// TwinCAT 3 PLC project SaftyPLC
// ProgramVersion: 3.1.4026.13
// libraries:
//   Tc2_Standard, * (Beckhoff Automation GmbH)
//   Tc2_System, * (Beckhoff Automation GmbH)
//   Tc2_Utilities, * (Beckhoff Automation GmbH)
//   Tc3_EventLogger, * (Beckhoff Automation GmbH)
//   Tc3_Module, * (Beckhoff Automation GmbH)
// project tree:
//   GVLs/ GVL_IO.TcGVL (not stored), GVL_Safety.TcGVL
//   / PlcTask.TcTTO
//   POUs/ MAIN.TcPOU
// real-time tasks:
//   TASK XTS Task: cycle T#500us, priority 1, ADS port 350
//   TASK Job Task: cycle default, priority 32
//   TASK MC-Task (MET): cycle T#2ms, priority 3, ADS port 521
//   TASK MC-Task (MPT): cycle T#10ms, priority 8, ADS port 531
//   TASK PlcTask: cycle T#500us, priority 20, ADS port 351
// motion (NC):
//   TASK NC-Task 1 SAF: cycle T#2ms, priority 4, ADS port 501
//   TASK NC-Task 1 SVB: cycle T#10ms, priority 9, ADS port 511
//   AXIS Axis 1 (id 1)
//     Velo: Maximum=4000
//     OtherSettings: AllowMotionCmdToSlave=true
//     encoder EncType=28
//       EncPara: MaxCount=#xffffffff
//     drive DrvType=22
//       DrvPara: MaxCount=#xffffffff, DriveControlDWord=#x00000100
//         Analog: VeloReferenz=4200, TorqueSetpointScale=10, ScaleFactorActTorque=0.1
//         TimeComp: TaskDelayCycles=1
//     controller CtrType=1
//       CtrPara: PriorControlFactor=1
//         Observer: BandWidth=20
// I/O:
//   DEVICE Device 8 (EtherCAT), AmsNetId 0.0.0.0.9.1
//     Box 77 (AT5100-0100) [AT5100-0100 XTS XL, TwinSAFE]
//       modules: Module 1 (SAFETY)
//     Box 78 (AT5100-0100) [AT5100-0100 XTS XL, TwinSAFE]
//       modules: Module 1 (SAFETY)
//     Box 79 (AT5100-0100) [AT5100-0100 XTS XL, TwinSAFE]
//       modules: Module 1 (SAFETY)
//     Box 80 (AT5100-0100) [AT5100-0100 XTS XL, TwinSAFE]
//       modules: Module 1 (SAFETY)
//     Box 81 (AT5100-0100) [AT5100-0100 XTS XL, TwinSAFE]
//       modules: Module 1 (SAFETY)
//     Box 18 (AT5100-0100) [AT5100-0100 XTS XL, TwinSAFE]
//       modules: Module 1 (SAFETY)
//     Box 19 (AT5100-0100) [AT5100-0100 XTS XL, TwinSAFE]
//       modules: Module 1 (SAFETY)
//     Box 20 (AT5100-0100) [AT5100-0100 XTS XL, TwinSAFE]
//       modules: Module 1 (SAFETY)
//     Box 21 (AT5100-0100) [AT5100-0100 XTS XL, TwinSAFE]
//       modules: Module 1 (SAFETY)
//     Box 22 (AT5100-0100) [AT5100-0100 XTS XL, TwinSAFE]
//       modules: Module 1 (SAFETY)
//   DEVICE Device 1 (EtherCAT), AmsNetId 0.0.0.0.2.1
//     Term 1 (EK1200) [EK1200-5000 EtherCAT Power supply (2A E-Bus)]
//       Term 2 (EL1809) [EL1809 16Ch. Dig. Input 24V, 3ms]
//       Term 3 (EL2809) [EL2809 16Ch. Dig. Output 24V, 0.5A]
//       Term 4 (EL1918) [EL1918, 8Ch. Safety Input 24V, TwinSAFE]
//         modules: Module 2 (FSLOGIC)
//       Term 5 (EK1110) [EK1110 EtherCAT extension]
//     Box 11 (Drive1211) [Drive1211]
//       modules: Module 1 (Standard Process Data)
//   DEVICE Device 2 (EtherCAT Automation Protocol), AmsNetId 0.0.0.0.3.1
//     Box 28 (Publisher)
//     Box 29 (Subscriber)
// variable links:
//   Device 1 (EtherCAT) <-> Device 2 (EtherCAT Automation Protocol)/Box 28 (Publisher)
//     Term 1 (EK1200)/Term 4 (EL1918)/ConnectionInputs/Message_144 TxPDO <-> Safety/Outputs/VarData
//   Device 1 (EtherCAT) <-> Device 2 (EtherCAT Automation Protocol)/Box 29 (Subscriber)
//     Term 1 (EK1200)/Term 4 (EL1918)/ConnectionOutputs/Message_144 RxPDO <-> Safety/Inputs/VarData
//   Device 2 (EtherCAT Automation Protocol) <-> MC Project IPC2/Groups/IPC 2 In Connection
//     Box 28 (Publisher)/MC Track - XL In Syst 2/Outputs/VarData <-> McToMc/ToNeighbourSystem
//     Box 29 (Subscriber)/MC Track - XL Out Syst 1/Inputs/VarData <-> McToMc/FromNeighbourSystem
//   Device 2 (EtherCAT Automation Protocol) <-> MC Project IPC2/Groups/IPC 2 Out Connection
//     Box 28 (Publisher)/MC Track - XL Out Syst 2/Outputs/VarData <-> McToMc/ToNeighbourSystem
//     Box 29 (Subscriber)/MC Track - XL In Syst 1/Inputs/VarData <-> McToMc/FromNeighbourSystem
//   Device 8 (EtherCAT) <-> Device 1 (EtherCAT)/Term 1 (EK1200)/Term 4 (EL1918)
//     Box 18 (AT5100-0100)/Module 1 (SAFETY)/SAFETY FSoE Connection 1 Receive Message/Message_4 <-> ConnectionInputs/Message_71 TxPDO
//     Box 19 (AT5100-0100)/Module 1 (SAFETY)/SAFETY FSoE Connection 1 Receive Message/Message_4 <-> ConnectionInputs/Message_76 TxPDO
//     Box 20 (AT5100-0100)/Module 1 (SAFETY)/SAFETY FSoE Connection 1 Receive Message/Message_4 <-> ConnectionInputs/Message_77 TxPDO
//     Box 21 (AT5100-0100)/Module 1 (SAFETY)/SAFETY FSoE Connection 1 Receive Message/Message_4 <-> ConnectionInputs/Message_78 TxPDO
//     Box 22 (AT5100-0100)/Module 1 (SAFETY)/SAFETY FSoE Connection 1 Receive Message/Message_4 <-> ConnectionInputs/Message_79 TxPDO
//     Box 77 (AT5100-0100)/Module 1 (SAFETY)/SAFETY FSoE Connection 1 Receive Message/Message_4 <-> ConnectionInputs/Message_134 TxPDO
//     Box 78 (AT5100-0100)/Module 1 (SAFETY)/SAFETY FSoE Connection 1 Receive Message/Message_4 <-> ConnectionInputs/Message_135 TxPDO
//     Box 79 (AT5100-0100)/Module 1 (SAFETY)/SAFETY FSoE Connection 1 Receive Message/Message_4 <-> ConnectionInputs/Message_136 TxPDO
//     Box 80 (AT5100-0100)/Module 1 (SAFETY)/SAFETY FSoE Connection 1 Receive Message/Message_4 <-> ConnectionInputs/Message_137 TxPDO
//     Box 81 (AT5100-0100)/Module 1 (SAFETY)/SAFETY FSoE Connection 1 Receive Message/Message_4 <-> ConnectionInputs/Message_138 TxPDO
//     Box 18 (AT5100-0100)/Module 1 (SAFETY)/SAFETY FSoE Connection 1 Send Message/Message_4 <-> ConnectionOutputs/Message_71 RxPDO
//     Box 19 (AT5100-0100)/Module 1 (SAFETY)/SAFETY FSoE Connection 1 Send Message/Message_4 <-> ConnectionOutputs/Message_76 RxPDO
//     Box 20 (AT5100-0100)/Module 1 (SAFETY)/SAFETY FSoE Connection 1 Send Message/Message_4 <-> ConnectionOutputs/Message_77 RxPDO
//     Box 21 (AT5100-0100)/Module 1 (SAFETY)/SAFETY FSoE Connection 1 Send Message/Message_4 <-> ConnectionOutputs/Message_78 RxPDO
//     Box 22 (AT5100-0100)/Module 1 (SAFETY)/SAFETY FSoE Connection 1 Send Message/Message_4 <-> ConnectionOutputs/Message_79 RxPDO
//     Box 77 (AT5100-0100)/Module 1 (SAFETY)/SAFETY FSoE Connection 1 Send Message/Message_4 <-> ConnectionOutputs/Message_134 RxPDO
//     Box 78 (AT5100-0100)/Module 1 (SAFETY)/SAFETY FSoE Connection 1 Send Message/Message_4 <-> ConnectionOutputs/Message_135 RxPDO
//     Box 79 (AT5100-0100)/Module 1 (SAFETY)/SAFETY FSoE Connection 1 Send Message/Message_4 <-> ConnectionOutputs/Message_136 RxPDO
//     Box 80 (AT5100-0100)/Module 1 (SAFETY)/SAFETY FSoE Connection 1 Send Message/Message_4 <-> ConnectionOutputs/Message_137 RxPDO
//     Box 81 (AT5100-0100)/Module 1 (SAFETY)/SAFETY FSoE Connection 1 Send Message/Message_4 <-> ConnectionOutputs/Message_138 RxPDO
//   MC Project IPC2/Axes/MC_Mover 01 IPC2 <-> MC Project IPC2/Axes/MC_Mover 01 IPC2/XConverter 01 IPC2
//     IoToMc/STD <-> OutputsToMC3/HWToMC3
//     McToIo/STD <-> InputsFromPlanarMover/MC3ToHW
//   MC Project IPC2/Axes/MC_Mover 02 IPC2 <-> MC Project IPC2/Axes/MC_Mover 02 IPC2/XConverter 02 IPC2
//     IoToMc/STD <-> OutputsToMC3/HWToMC3
//     McToIo/STD <-> InputsFromPlanarMover/MC3ToHW
//   MC Project IPC2/Axes/MC_Mover 03 IPC2 <-> MC Project IPC2/Axes/MC_Mover 03 IPC2/XConverter 03 IPC2
//     IoToMc/STD <-> OutputsToMC3/HWToMC3
//     McToIo/STD <-> InputsFromPlanarMover/MC3ToHW
//   MC Project IPC2/Axes/MC_Mover 04 IPC2 <-> MC Project IPC2/Axes/MC_Mover 04 IPC2/XConverter 04 IPC2
//     IoToMc/STD <-> OutputsToMC3/HWToMC3
//     McToIo/STD <-> InputsFromPlanarMover/MC3ToHW
//   MC Project IPC2/Axes/MC_Mover 05 IPC2 <-> MC Project IPC2/Axes/MC_Mover 05 IPC2/XConverter 05 IPC2
//     IoToMc/STD <-> OutputsToMC3/HWToMC3
//     McToIo/STD <-> InputsFromPlanarMover/MC3ToHW
//   MC Project IPC2/Axes/MC_Mover 06 IPC2 <-> MC Project IPC2/Axes/MC_Mover 06 IPC2/XConverter 06 IPC2
//     IoToMc/STD <-> OutputsToMC3/HWToMC3
//     McToIo/STD <-> InputsFromPlanarMover/MC3ToHW
//   MC Project IPC2/Axes/MC_Mover 07 IPC2 <-> MC Project IPC2/Axes/MC_Mover 07 IPC2/XConverter 07 IPC2
//     IoToMc/STD <-> OutputsToMC3/HWToMC3
//     McToIo/STD <-> InputsFromPlanarMover/MC3ToHW
//   MC Project IPC2/Axes/MC_Mover 08 IPC2 <-> MC Project IPC2/Axes/MC_Mover 08 IPC2/XConverter 08 IPC2
//     IoToMc/STD <-> OutputsToMC3/HWToMC3
//     McToIo/STD <-> InputsFromPlanarMover/MC3ToHW
//   MC Project IPC2/Axes/MC_Mover 09 IPC2 <-> MC Project IPC2/Axes/MC_Mover 09 IPC2/XConverter 09 IPC2
//     IoToMc/STD <-> OutputsToMC3/HWToMC3
//     McToIo/STD <-> InputsFromPlanarMover/MC3ToHW
//   MC Project IPC2/Axes/MC_Mover 10 IPC2 <-> MC Project IPC2/Axes/MC_Mover 10 IPC2/XConverter 10 IPC2
//     IoToMc/STD <-> OutputsToMC3/HWToMC3
//     McToIo/STD <-> InputsFromPlanarMover/MC3ToHW
//   MC Project IPC2/Axes/MC_Mover 11 IPC2 <-> MC Project IPC2/Axes/MC_Mover 11 IPC2/XConverter 11 IPC2
//     IoToMc/STD <-> OutputsToMC3/HWToMC3
//     McToIo/STD <-> InputsFromPlanarMover/MC3ToHW
//   MC Project IPC2/Axes/MC_Mover 12 IPC2 <-> MC Project IPC2/Axes/MC_Mover 12 IPC2/XConverter 12 IPC2
//     IoToMc/STD <-> OutputsToMC3/HWToMC3
//     McToIo/STD <-> InputsFromPlanarMover/MC3ToHW
//   MC3_Multi_IPC2/MC3_Multi_IPC2 Instance <-> Device 2 (EtherCAT Automation Protocol)/Box 29 (Subscriber)
//     PlcTask Inputs/GVL_DataExchange.Dynamics <-> Command/Inputs/VarData/Dynamics
//   MC3_Multi_IPC2/MC3_Multi_IPC2 Instance <-> MC Project IPC2/Axes/MC_Mover 01 IPC2
//     PlcTask Inputs/GVL_MC.fbMover[1].fbPlanarMover.MCTOPLC/ACT <-> McToPlc/ACT
//     PlcTask Inputs/GVL_MC.fbMover[1].fbPlanarMover.MCTOPLC/COORDMODE <-> McToPlc/COORDMODE
//     PlcTask Inputs/GVL_MC.fbMover[1].fbPlanarMover.MCTOPLC/SET <-> McToPlc/SET
//     PlcTask Inputs/GVL_MC.fbMover[1].fbPlanarMover.MCTOPLC/SETONTRACK <-> McToPlc/SETONTRACK
//     PlcTask Inputs/GVL_MC.fbMover[1].fbPlanarMover.MCTOPLC/STD <-> McToPlc/STD
//     PlcTask Outputs/GVL_MC.fbMover[1].fbPlanarMover.PLCTOMC/STD <-> PlcToMc/STD
//   MC3_Multi_IPC2/MC3_Multi_IPC2 Instance <-> MC Project IPC2/Axes/MC_Mover 02 IPC2
//     PlcTask Inputs/GVL_MC.fbMover[2].fbPlanarMover.MCTOPLC/ACT <-> McToPlc/ACT
//     PlcTask Inputs/GVL_MC.fbMover[2].fbPlanarMover.MCTOPLC/COORDMODE <-> McToPlc/COORDMODE
//     PlcTask Inputs/GVL_MC.fbMover[2].fbPlanarMover.MCTOPLC/SET <-> McToPlc/SET
//     PlcTask Inputs/GVL_MC.fbMover[2].fbPlanarMover.MCTOPLC/SETONTRACK <-> McToPlc/SETONTRACK
//     PlcTask Inputs/GVL_MC.fbMover[2].fbPlanarMover.MCTOPLC/STD <-> McToPlc/STD
//     PlcTask Outputs/GVL_MC.fbMover[2].fbPlanarMover.PLCTOMC/STD <-> PlcToMc/STD
//   MC3_Multi_IPC2/MC3_Multi_IPC2 Instance <-> MC Project IPC2/Axes/MC_Mover 03 IPC2
//     PlcTask Inputs/GVL_MC.fbMover[3].fbPlanarMover.MCTOPLC/ACT <-> McToPlc/ACT
//     PlcTask Inputs/GVL_MC.fbMover[3].fbPlanarMover.MCTOPLC/COORDMODE <-> McToPlc/COORDMODE
//     PlcTask Inputs/GVL_MC.fbMover[3].fbPlanarMover.MCTOPLC/SET <-> McToPlc/SET
//     PlcTask Inputs/GVL_MC.fbMover[3].fbPlanarMover.MCTOPLC/SETONTRACK <-> McToPlc/SETONTRACK
//     PlcTask Inputs/GVL_MC.fbMover[3].fbPlanarMover.MCTOPLC/STD <-> McToPlc/STD
//     PlcTask Outputs/GVL_MC.fbMover[3].fbPlanarMover.PLCTOMC/STD <-> PlcToMc/STD
//   MC3_Multi_IPC2/MC3_Multi_IPC2 Instance <-> MC Project IPC2/Axes/MC_Mover 04 IPC2
//     PlcTask Inputs/GVL_MC.fbMover[4].fbPlanarMover.MCTOPLC/ACT <-> McToPlc/ACT
//     PlcTask Inputs/GVL_MC.fbMover[4].fbPlanarMover.MCTOPLC/COORDMODE <-> McToPlc/COORDMODE
//     PlcTask Inputs/GVL_MC.fbMover[4].fbPlanarMover.MCTOPLC/SET <-> McToPlc/SET
//     PlcTask Inputs/GVL_MC.fbMover[4].fbPlanarMover.MCTOPLC/SETONTRACK <-> McToPlc/SETONTRACK
//     PlcTask Inputs/GVL_MC.fbMover[4].fbPlanarMover.MCTOPLC/STD <-> McToPlc/STD
//     PlcTask Outputs/GVL_MC.fbMover[4].fbPlanarMover.PLCTOMC/STD <-> PlcToMc/STD
//   MC3_Multi_IPC2/MC3_Multi_IPC2 Instance <-> MC Project IPC2/Axes/MC_Mover 05 IPC2
//     PlcTask Inputs/GVL_MC.fbMover[5].fbPlanarMover.MCTOPLC/ACT <-> McToPlc/ACT
//     PlcTask Inputs/GVL_MC.fbMover[5].fbPlanarMover.MCTOPLC/COORDMODE <-> McToPlc/COORDMODE
//     PlcTask Inputs/GVL_MC.fbMover[5].fbPlanarMover.MCTOPLC/SET <-> McToPlc/SET
//     PlcTask Inputs/GVL_MC.fbMover[5].fbPlanarMover.MCTOPLC/SETONTRACK <-> McToPlc/SETONTRACK
//     PlcTask Inputs/GVL_MC.fbMover[5].fbPlanarMover.MCTOPLC/STD <-> McToPlc/STD
//     PlcTask Outputs/GVL_MC.fbMover[5].fbPlanarMover.PLCTOMC/STD <-> PlcToMc/STD
//   MC3_Multi_IPC2/MC3_Multi_IPC2 Instance <-> MC Project IPC2/Axes/MC_Mover 06 IPC2
//     PlcTask Inputs/GVL_MC.fbMover[6].fbPlanarMover.MCTOPLC/ACT <-> McToPlc/ACT
//     PlcTask Inputs/GVL_MC.fbMover[6].fbPlanarMover.MCTOPLC/COORDMODE <-> McToPlc/COORDMODE
//     PlcTask Inputs/GVL_MC.fbMover[6].fbPlanarMover.MCTOPLC/SET <-> McToPlc/SET
//     PlcTask Inputs/GVL_MC.fbMover[6].fbPlanarMover.MCTOPLC/SETONTRACK <-> McToPlc/SETONTRACK
//     PlcTask Inputs/GVL_MC.fbMover[6].fbPlanarMover.MCTOPLC/STD <-> McToPlc/STD
//     PlcTask Outputs/GVL_MC.fbMover[6].fbPlanarMover.PLCTOMC/STD <-> PlcToMc/STD
//   MC3_Multi_IPC2/MC3_Multi_IPC2 Instance <-> MC Project IPC2/Axes/MC_Mover 07 IPC2
//     PlcTask Inputs/GVL_MC.fbMover[7].fbPlanarMover.MCTOPLC/ACT <-> McToPlc/ACT
//     PlcTask Inputs/GVL_MC.fbMover[7].fbPlanarMover.MCTOPLC/COORDMODE <-> McToPlc/COORDMODE
//     PlcTask Inputs/GVL_MC.fbMover[7].fbPlanarMover.MCTOPLC/SET <-> McToPlc/SET
//     PlcTask Inputs/GVL_MC.fbMover[7].fbPlanarMover.MCTOPLC/SETONTRACK <-> McToPlc/SETONTRACK
//     PlcTask Inputs/GVL_MC.fbMover[7].fbPlanarMover.MCTOPLC/STD <-> McToPlc/STD
//     PlcTask Outputs/GVL_MC.fbMover[7].fbPlanarMover.PLCTOMC/STD <-> PlcToMc/STD
//   MC3_Multi_IPC2/MC3_Multi_IPC2 Instance <-> MC Project IPC2/Axes/MC_Mover 08 IPC2
//     PlcTask Inputs/GVL_MC.fbMover[8].fbPlanarMover.MCTOPLC/ACT <-> McToPlc/ACT
//     PlcTask Inputs/GVL_MC.fbMover[8].fbPlanarMover.MCTOPLC/COORDMODE <-> McToPlc/COORDMODE
//     PlcTask Inputs/GVL_MC.fbMover[8].fbPlanarMover.MCTOPLC/SET <-> McToPlc/SET
//     PlcTask Inputs/GVL_MC.fbMover[8].fbPlanarMover.MCTOPLC/SETONTRACK <-> McToPlc/SETONTRACK
//     PlcTask Inputs/GVL_MC.fbMover[8].fbPlanarMover.MCTOPLC/STD <-> McToPlc/STD
//     PlcTask Outputs/GVL_MC.fbMover[8].fbPlanarMover.PLCTOMC/STD <-> PlcToMc/STD
//   MC3_Multi_IPC2/MC3_Multi_IPC2 Instance <-> MC Project IPC2/Axes/MC_Mover 09 IPC2
//     PlcTask Inputs/GVL_MC.fbMover[9].fbPlanarMover.MCTOPLC/ACT <-> McToPlc/ACT
//     PlcTask Inputs/GVL_MC.fbMover[9].fbPlanarMover.MCTOPLC/COORDMODE <-> McToPlc/COORDMODE
//     PlcTask Inputs/GVL_MC.fbMover[9].fbPlanarMover.MCTOPLC/SET <-> McToPlc/SET
//     PlcTask Inputs/GVL_MC.fbMover[9].fbPlanarMover.MCTOPLC/SETONTRACK <-> McToPlc/SETONTRACK
//     PlcTask Inputs/GVL_MC.fbMover[9].fbPlanarMover.MCTOPLC/STD <-> McToPlc/STD
//     PlcTask Outputs/GVL_MC.fbMover[9].fbPlanarMover.PLCTOMC/STD <-> PlcToMc/STD
//   MC3_Multi_IPC2/MC3_Multi_IPC2 Instance <-> MC Project IPC2/Axes/MC_Mover 10 IPC2
//     PlcTask Inputs/GVL_MC.fbMover[10].fbPlanarMover.MCTOPLC/ACT <-> McToPlc/ACT
//     PlcTask Inputs/GVL_MC.fbMover[10].fbPlanarMover.MCTOPLC/COORDMODE <-> McToPlc/COORDMODE
//     PlcTask Inputs/GVL_MC.fbMover[10].fbPlanarMover.MCTOPLC/SET <-> McToPlc/SET
//     PlcTask Inputs/GVL_MC.fbMover[10].fbPlanarMover.MCTOPLC/SETONTRACK <-> McToPlc/SETONTRACK
//     PlcTask Inputs/GVL_MC.fbMover[10].fbPlanarMover.MCTOPLC/STD <-> McToPlc/STD
//     PlcTask Outputs/GVL_MC.fbMover[10].fbPlanarMover.PLCTOMC/STD <-> PlcToMc/STD
//   MC3_Multi_IPC2/MC3_Multi_IPC2 Instance <-> MC Project IPC2/Axes/MC_Mover 11 IPC2
//     PlcTask Inputs/GVL_MC.fbMover[11].fbPlanarMover.MCTOPLC/ACT <-> McToPlc/ACT
//     PlcTask Inputs/GVL_MC.fbMover[11].fbPlanarMover.MCTOPLC/COORDMODE <-> McToPlc/COORDMODE
//     PlcTask Inputs/GVL_MC.fbMover[11].fbPlanarMover.MCTOPLC/SET <-> McToPlc/SET
//     PlcTask Inputs/GVL_MC.fbMover[11].fbPlanarMover.MCTOPLC/SETONTRACK <-> McToPlc/SETONTRACK
//     PlcTask Inputs/GVL_MC.fbMover[11].fbPlanarMover.MCTOPLC/STD <-> McToPlc/STD
//     PlcTask Outputs/GVL_MC.fbMover[11].fbPlanarMover.PLCTOMC/STD <-> PlcToMc/STD
//   MC3_Multi_IPC2/MC3_Multi_IPC2 Instance <-> MC Project IPC2/Axes/MC_Mover 12 IPC2
//     PlcTask Inputs/GVL_MC.fbMover[12].fbPlanarMover.MCTOPLC/ACT <-> McToPlc/ACT
//     PlcTask Inputs/GVL_MC.fbMover[12].fbPlanarMover.MCTOPLC/COORDMODE <-> McToPlc/COORDMODE
//     PlcTask Inputs/GVL_MC.fbMover[12].fbPlanarMover.MCTOPLC/SET <-> McToPlc/SET
//     PlcTask Inputs/GVL_MC.fbMover[12].fbPlanarMover.MCTOPLC/SETONTRACK <-> McToPlc/SETONTRACK
//     PlcTask Inputs/GVL_MC.fbMover[12].fbPlanarMover.MCTOPLC/STD <-> McToPlc/STD
//     PlcTask Outputs/GVL_MC.fbMover[12].fbPlanarMover.PLCTOMC/STD <-> PlcToMc/STD
//   MC3_Multi_IPC2/MC3_Multi_IPC2 Instance <-> MC Project IPC2/Groups/IPC 2 In Connection
//     PlcTask Inputs/GVL_MC.EnterSystem.MCTOPLC_STD <-> McToPlc/STD
//   MC3_Multi_IPC2/MC3_Multi_IPC2 Instance <-> MC Project IPC2/Groups/IPC 2 Out Connection
//     PlcTask Inputs/GVL_MC.ExitSystem.MCTOPLC_STD <-> McToPlc/STD
//   MC3_Multi_IPC2/MC3_Multi_IPC2 Instance <-> MC Project IPC2/Groups/McTrack1
//     PlcTask Inputs/GVL_MC.aMcTracks[1].MCTOPLC_STD <-> McToPlc/STD
//   SaftyPLC/SaftyPLC Instance <-> Device 1 (EtherCAT)/Box 11 (Drive1211)
//     PlcTask Inputs/GVL_IO.StatusDrive1121 <-> Module 1 (Standard Process Data)/TxPDO1Map entries/Statusword
//     PlcTask Inputs/GVL_IO.VoltageAct <-> Module 1 (Standard Process Data)/TxPDO1Map entries/Zwischenkreisspannung
//     PlcTask Outputs/GVL_IO.ControlDrive1121 <-> Module 1 (Standard Process Data)/RxPDO1Map entries/Controlword
//     PlcTask Outputs/GVL_IO.VoltageSet <-> Module 1 (Standard Process Data)/RxPDO1Map entries/Zwischenkreisspannung Soll
//   SaftyPLC/SaftyPLC Instance <-> Device 1 (EtherCAT)/Term 1 (EK1200)/Term 2 (EL1809)
//     PlcTask Inputs/GVL_Safety.HWReset <-> Channel 16/Input
//     PlcTask Inputs/GVL_Safety.HWStart <-> Channel 14/Input
//     PlcTask Inputs/GVL_Safety.HWStop <-> Channel 15/Input
//   SaftyPLC/SaftyPLC Instance <-> Device 1 (EtherCAT)/Term 1 (EK1200)/Term 3 (EL2809)
//     PlcTask Outputs/GVL_Safety.HWSafetyOk <-> Channel 14/Output
//     PlcTask Outputs/GVL_Safety.HWerror <-> Channel 15/Output
//   SaftyPLC/SaftyPLC Instance <-> Device 1 (EtherCAT)/Term 1 (EK1200)/Term 4 (EL1918)
//     PlcTask Inputs/GVL_Safety.SaeftyOk <-> StandardInputs/Standard Out Var 139
//     PlcTask Outputs/GVL_Safety.Reset <-> StandardOutputs/Standard In Var 1
//     PlcTask Outputs/GVL_Safety.Run <-> StandardOutputs/Standard In Var 2
//     PlcTask Outputs/GVL_Safety.Start <-> StandardOutputs/Standard In Var 140
//     PlcTask Outputs/GVL_Safety.Start <-> StandardOutputs/Standard In Var 75
//   SaftyPLC/SaftyPLC Instance <-> Device 2 (EtherCAT Automation Protocol)/Box 29 (Subscriber)
//     PlcTask Inputs/GVL_Safety.MasterReset <-> Command/Inputs/VarData/Reset
//     PlcTask Inputs/GVL_Safety.SafetyInRun <-> Command/Inputs/VarData/Run
//   SaftyPLC/SaftyPLC Instance <-> Device 8 (EtherCAT)/Box 18 (AT5100-0100)
//     PlcTask Outputs/GVL_Safety.Reset <-> Module 1 (SAFETY)/SAFETY Standard Outputdata/Standard In Var 1
//     PlcTask Outputs/GVL_Safety.Run <-> Module 1 (SAFETY)/SAFETY Standard Outputdata/Standard In Var 2
//   SaftyPLC/SaftyPLC Instance <-> Device 8 (EtherCAT)/Box 19 (AT5100-0100)
//     PlcTask Outputs/GVL_Safety.Reset <-> Module 1 (SAFETY)/SAFETY Standard Outputdata/Standard In Var 1
//     PlcTask Outputs/GVL_Safety.Run <-> Module 1 (SAFETY)/SAFETY Standard Outputdata/Standard In Var 2
//   SaftyPLC/SaftyPLC Instance <-> Device 8 (EtherCAT)/Box 20 (AT5100-0100)
//     PlcTask Outputs/GVL_Safety.Reset <-> Module 1 (SAFETY)/SAFETY Standard Outputdata/Standard In Var 1
//     PlcTask Outputs/GVL_Safety.Run <-> Module 1 (SAFETY)/SAFETY Standard Outputdata/Standard In Var 2
//   SaftyPLC/SaftyPLC Instance <-> Device 8 (EtherCAT)/Box 21 (AT5100-0100)
//     PlcTask Outputs/GVL_Safety.Reset <-> Module 1 (SAFETY)/SAFETY Standard Outputdata/Standard In Var 1
//     PlcTask Outputs/GVL_Safety.Run <-> Module 1 (SAFETY)/SAFETY Standard Outputdata/Standard In Var 2
//   SaftyPLC/SaftyPLC Instance <-> Device 8 (EtherCAT)/Box 22 (AT5100-0100)
//     PlcTask Outputs/GVL_Safety.Reset <-> Module 1 (SAFETY)/SAFETY Standard Outputdata/Standard In Var 1
//     PlcTask Outputs/GVL_Safety.Run <-> Module 1 (SAFETY)/SAFETY Standard Outputdata/Standard In Var 2
//   SaftyPLC/SaftyPLC Instance <-> Device 8 (EtherCAT)/Box 77 (AT5100-0100)
//     PlcTask Outputs/GVL_Safety.Reset <-> Module 1 (SAFETY)/SAFETY Standard Outputdata/Standard In Var 1
//     PlcTask Outputs/GVL_Safety.Run <-> Module 1 (SAFETY)/SAFETY Standard Outputdata/Standard In Var 2
//   SaftyPLC/SaftyPLC Instance <-> Device 8 (EtherCAT)/Box 78 (AT5100-0100)
//     PlcTask Outputs/GVL_Safety.Reset <-> Module 1 (SAFETY)/SAFETY Standard Outputdata/Standard In Var 1
//     PlcTask Outputs/GVL_Safety.Run <-> Module 1 (SAFETY)/SAFETY Standard Outputdata/Standard In Var 2
//   SaftyPLC/SaftyPLC Instance <-> Device 8 (EtherCAT)/Box 79 (AT5100-0100)
//     PlcTask Outputs/GVL_Safety.Reset <-> Module 1 (SAFETY)/SAFETY Standard Outputdata/Standard In Var 1
//     PlcTask Outputs/GVL_Safety.Run <-> Module 1 (SAFETY)/SAFETY Standard Outputdata/Standard In Var 2
//   SaftyPLC/SaftyPLC Instance <-> Device 8 (EtherCAT)/Box 80 (AT5100-0100)
//     PlcTask Outputs/GVL_Safety.Reset <-> Module 1 (SAFETY)/SAFETY Standard Outputdata/Standard In Var 1
//     PlcTask Outputs/GVL_Safety.Run <-> Module 1 (SAFETY)/SAFETY Standard Outputdata/Standard In Var 2
//   SaftyPLC/SaftyPLC Instance <-> Device 8 (EtherCAT)/Box 81 (AT5100-0100)
//     PlcTask Outputs/GVL_Safety.Reset <-> Module 1 (SAFETY)/SAFETY Standard Outputdata/Standard In Var 1
//     PlcTask Outputs/GVL_Safety.Run <-> Module 1 (SAFETY)/SAFETY Standard Outputdata/Standard In Var 2
//   (this object) <-> TcCOM Objects/XTS ProcessingUnit 2/XL Part Main/XL Module 10
//     Box 19 (AT5100-0100)/DRV Commutation angle/Commutation angle <-> Data Pointer/CommutationAngle
//     Box 19 (AT5100-0100)/DRV Controlword/Controlword <-> Data Pointer/Control
//     Box 19 (AT5100-0100)/DRV Statusword/Statusword <-> Data Pointer/Status
//     Box 19 (AT5100-0100)/DRV Target torque/Target torque <-> Data Pointer/Torque
//     Box 19 (AT5100-0100)/DRV Torque actual value/Torque actual value <-> Data Pointer/ActTorque
//     Box 19 (AT5100-0100)/XFB Inputs/Data <-> Data Pointer/HallSensorValues
//   (this object) <-> TcCOM Objects/XTS ProcessingUnit 2/XL Part Main/XL Module 11
//     Box 20 (AT5100-0100)/DRV Commutation angle/Commutation angle <-> Data Pointer/CommutationAngle
//     Box 20 (AT5100-0100)/DRV Controlword/Controlword <-> Data Pointer/Control
//     Box 20 (AT5100-0100)/DRV Statusword/Statusword <-> Data Pointer/Status
//     Box 20 (AT5100-0100)/DRV Target torque/Target torque <-> Data Pointer/Torque
//     Box 20 (AT5100-0100)/DRV Torque actual value/Torque actual value <-> Data Pointer/ActTorque
//     Box 20 (AT5100-0100)/XFB Inputs/Data <-> Data Pointer/HallSensorValues
//   (this object) <-> TcCOM Objects/XTS ProcessingUnit 2/XL Part Main/XL Module 12
//     Box 21 (AT5100-0100)/DRV Commutation angle/Commutation angle <-> Data Pointer/CommutationAngle
//     Box 21 (AT5100-0100)/DRV Controlword/Controlword <-> Data Pointer/Control
//     Box 21 (AT5100-0100)/DRV Statusword/Statusword <-> Data Pointer/Status
//     Box 21 (AT5100-0100)/DRV Target torque/Target torque <-> Data Pointer/Torque
//     Box 21 (AT5100-0100)/DRV Torque actual value/Torque actual value <-> Data Pointer/ActTorque
//     Box 21 (AT5100-0100)/XFB Inputs/Data <-> Data Pointer/HallSensorValues
//   (this object) <-> TcCOM Objects/XTS ProcessingUnit 2/XL Part Main/XL Module 13
//     Box 22 (AT5100-0100)/DRV Commutation angle/Commutation angle <-> Data Pointer/CommutationAngle
//     Box 22 (AT5100-0100)/DRV Controlword/Controlword <-> Data Pointer/Control
//     Box 22 (AT5100-0100)/DRV Statusword/Statusword <-> Data Pointer/Status
//     Box 22 (AT5100-0100)/DRV Target torque/Target torque <-> Data Pointer/Torque
//     Box 22 (AT5100-0100)/DRV Torque actual value/Torque actual value <-> Data Pointer/ActTorque
//     Box 22 (AT5100-0100)/XFB Inputs/Data <-> Data Pointer/HallSensorValues
//   (this object) <-> TcCOM Objects/XTS ProcessingUnit 2/XL Part Main/XL Module 4
//     Box 77 (AT5100-0100)/DRV Commutation angle/Commutation angle <-> Data Pointer/CommutationAngle
//     Box 77 (AT5100-0100)/DRV Controlword/Controlword <-> Data Pointer/Control
//     Box 77 (AT5100-0100)/DRV Statusword/Statusword <-> Data Pointer/Status
//     Box 77 (AT5100-0100)/DRV Target torque/Target torque <-> Data Pointer/Torque
//     Box 77 (AT5100-0100)/DRV Torque actual value/Torque actual value <-> Data Pointer/ActTorque
//     Box 77 (AT5100-0100)/XFB Inputs/Data <-> Data Pointer/HallSensorValues
//   (this object) <-> TcCOM Objects/XTS ProcessingUnit 2/XL Part Main/XL Module 5
//     Box 78 (AT5100-0100)/DRV Commutation angle/Commutation angle <-> Data Pointer/CommutationAngle
//     Box 78 (AT5100-0100)/DRV Controlword/Controlword <-> Data Pointer/Control
//     Box 78 (AT5100-0100)/DRV Statusword/Statusword <-> Data Pointer/Status
//     Box 78 (AT5100-0100)/DRV Target torque/Target torque <-> Data Pointer/Torque
//     Box 78 (AT5100-0100)/DRV Torque actual value/Torque actual value <-> Data Pointer/ActTorque
//     Box 78 (AT5100-0100)/XFB Inputs/Data <-> Data Pointer/HallSensorValues
//   (this object) <-> TcCOM Objects/XTS ProcessingUnit 2/XL Part Main/XL Module 6
//     Box 79 (AT5100-0100)/DRV Commutation angle/Commutation angle <-> Data Pointer/CommutationAngle
//     Box 79 (AT5100-0100)/DRV Controlword/Controlword <-> Data Pointer/Control
//     Box 79 (AT5100-0100)/DRV Statusword/Statusword <-> Data Pointer/Status
//     Box 79 (AT5100-0100)/DRV Target torque/Target torque <-> Data Pointer/Torque
//     Box 79 (AT5100-0100)/DRV Torque actual value/Torque actual value <-> Data Pointer/ActTorque
//     Box 79 (AT5100-0100)/XFB Inputs/Data <-> Data Pointer/HallSensorValues
//   (this object) <-> TcCOM Objects/XTS ProcessingUnit 2/XL Part Main/XL Module 7
//     Box 80 (AT5100-0100)/DRV Commutation angle/Commutation angle <-> Data Pointer/CommutationAngle
//     Box 80 (AT5100-0100)/DRV Controlword/Controlword <-> Data Pointer/Control
//     Box 80 (AT5100-0100)/DRV Statusword/Statusword <-> Data Pointer/Status
//     Box 80 (AT5100-0100)/DRV Target torque/Target torque <-> Data Pointer/Torque
//     Box 80 (AT5100-0100)/DRV Torque actual value/Torque actual value <-> Data Pointer/ActTorque
//     Box 80 (AT5100-0100)/XFB Inputs/Data <-> Data Pointer/HallSensorValues
//   (this object) <-> TcCOM Objects/XTS ProcessingUnit 2/XL Part Main/XL Module 8
//     Box 81 (AT5100-0100)/DRV Commutation angle/Commutation angle <-> Data Pointer/CommutationAngle
//     Box 81 (AT5100-0100)/DRV Controlword/Controlword <-> Data Pointer/Control
//     Box 81 (AT5100-0100)/DRV Statusword/Statusword <-> Data Pointer/Status
//     Box 81 (AT5100-0100)/DRV Target torque/Target torque <-> Data Pointer/Torque
//     Box 81 (AT5100-0100)/DRV Torque actual value/Torque actual value <-> Data Pointer/ActTorque
//     Box 81 (AT5100-0100)/XFB Inputs/Data <-> Data Pointer/HallSensorValues
//   (this object) <-> TcCOM Objects/XTS ProcessingUnit 2/XL Part Main/XL Module 9
//     Box 18 (AT5100-0100)/DRV Commutation angle/Commutation angle <-> Data Pointer/CommutationAngle
//     Box 18 (AT5100-0100)/DRV Controlword/Controlword <-> Data Pointer/Control
//     Box 18 (AT5100-0100)/DRV Statusword/Statusword <-> Data Pointer/Status
//     Box 18 (AT5100-0100)/DRV Target torque/Target torque <-> Data Pointer/Torque
//     Box 18 (AT5100-0100)/DRV Torque actual value/Torque actual value <-> Data Pointer/ActTorque
//     Box 18 (AT5100-0100)/XFB Inputs/Data <-> Data Pointer/HallSensorValues

CONFIGURATION SaftyPLC
    RESOURCE PLC ON TwinCAT3
        TASK PlcTask(INTERVAL := T#500us, PRIORITY := 20);
        PROGRAM MAIN WITH PlcTask : MAIN;
    END_RESOURCE
END_CONFIGURATION

// ---- GVLs/GVL_Safety.TcGVL
{attribute 'qualified_only'}
VAR_GLOBAL
	Run			AT%Q* : BOOL := TRUE;
	Start		AT%Q* : BOOL := TRUE;
	Reset		AT%Q* : BOOL;
	MasterStart		AT%I* : BOOL;
	MasterReset		AT%I* : BOOL;
	
	
	SafetyInRun	AT%I* : BOOL;
	SaeftyOk 	AT%I* : BOOL;
	
	HWStart		AT%I* : BOOL;
	HWStop		AT%I* : BOOL;
	HWReset		AT%I* : BOOL;
	
	HWerror		AT%Q* : BOOL;
	HWSafetyOk	AT%Q* : BOOL;
	
END_VAR

// ---- POUs/MAIN.TcPOU
PROGRAM MAIN
VAR
	nCase 					: INT;
	HwStart 		AT%I* 	: BOOL;
	HwStop  		AT%I* 	: BOOL;
	HwReset 		AT%I* 	: BOOL;
	xOn 			AT%Q* 	: BOOL;
	xRequestReset 	AT%Q* 	: BOOL;
	xError 			AT%Q* 	: BOOL;
		
	VoltageSP 			  	: LREAL := 300;
	rTrigSwitchon 		  	: R_trig;
	fTrigSwitchOff		  	: F_trig;
	Chargtimer 				: ton;
	
	SwitchOn				: BOOL;
	
	TcRestart : TC_Restart;
	Restart : BOOL;
	busy : BOOL;

END_VAR



IF GVL_Safety.HWStart OR GVL_Safety.MasterStart THEN
	GVL_Safety.Run  := TRUE;
	GVL_Safety.Start := TRUE;
END_IF

IF  NOT GVL_Safety.HWStop THEN
	GVL_Safety.Run  := FALSE;
	GVL_Safety.Start := FALSE;
END_IF
		


IF gvl_safety.SaeftyOk THEN
	gvl_safety.HWSafetyOk := TRUE;
ELSE	
	gvl_safety.HWSafetyOk := FALSE;
END_IF

IF NOT gvl_safety.SafetyInRun THEN
	gvl_safety.HWerror := TRUE;
ELSE	
	gvl_safety.HWerror := FALSE;
END_IF

rTrigSwitchon(clk := HwStart );
fTrigSwitchOff(clk:= HwStop );


 Chargtimer(in := SwitchOn ,pt := T#1M, q=>GVL_IO.ChargingResistor);

IF rTrigSwitchon.Q THEN
	GVL_IO.VoltageSet := GVL_IO.VoltageAct;
	SwitchOn := TRUE;
ELSIF fTrigSwitchOff.Q THEN
	SwitchOn := FALSE;
	GVL_IO.VoltageSet :=   0;
END_IF



IF (VoltageSP-2) > GVL_IO.VoltageAct AND  GVL_IO.Voltageset <VoltageSP AND SwitchOn THEN
	GVL_IO.VoltageSet := GVL_IO.VoltageSet +0.1;
END_IF



IF GVL_IO.hwReset OR HwReset OR GVL_Safety.MasterReset THEN
	GVL_IO.ControlDrive1121 := 16#FF;
	GVL_Safety.Reset := TRUE;
ELSE 	
	GVL_IO.ControlDrive1121 := 16#0;
	GVL_Safety.Reset := FALSE;
END_IF

TcRestart(
	NETID:= , 
	RESTART:=Restart , 
	TMOUT:= , 
	BUSY=> , 
	ERR=> , 
	ERRID=> );

END_PROGRAM
